GLOBALCONSTANTS Filter (* Global constants *)
  (* Standard: 61499-1 *)
  (* Version 1.0, 2025-10-19, franz *)
  PACKAGE uebungen;
  IMPORT isobus::pgn::NAMEFIELD_T;
  VAR_GLOBAL CONSTANT
    VT_ADD : isobus::pgn::NAMEFIELD_T := (bSelfConf := FALSE, bIndGroup := 0, bDevClassInst := 0, bDevClass := 0,    bReserved := FALSE, bFunction := 29, bFunctionInst := 0, bEcuInstance := 0, wManufCode := 0,    dwIdentNumb := 0);
    VT_FLT : isobus::pgn::NAMEFIELD_T := (bSelfConf := FALSE, bIndGroup := 0, bDevClassInst := 0, bDevClass := 0,    bReserved := FALSE, bFunction := 16#FF, bFunctionInst := 0, bEcuInstance := 0, wManufCode := 0,    dwIdentNumb := 0);
    FLT_ALL_PASS : isobus::pgn::NAMEFIELD_T := (bSelfConf := FALSE, bIndGroup := 0, bDevClassInst := 0, bDevClass := 0,    bReserved := FALSE, bFunction := 0, bFunctionInst := 0, bEcuInstance := 0, wManufCode := 0,    dwIdentNumb := 0);
    PEAK_ADD : isobus::pgn::NAMEFIELD_T := (bSelfConf := FALSE, bIndGroup := 4, bDevClassInst := 0, bDevClass := 0,    bReserved := FALSE, bFunction := 99, bFunctionInst := 9, bEcuInstance := 0, wManufCode := 0,    dwIdentNumb := 0);
    PEAK_FLT : isobus::pgn::NAMEFIELD_T := (bSelfConf := FALSE, bIndGroup := 16#FF, bDevClassInst := 0, bDevClass := 0,    bReserved := FALSE, bFunction := 16#FF, bFunctionInst := 16#FF, bEcuInstance := 0, wManufCode := 0,    dwIdentNumb := 0);
  END_VAR
END_GLOBALCONSTANTS
